// TwinCAT 3 PLC project Library
// Title: lcls-twincat-motion
// Company: SLAC
// ProjectVersion: 0.0.0
// ProgramVersion: 3.1.4026.17
// libraries:
//   LCLS General, * (SLAC)
//   lcls-twincat-math, * (SLAC - LCLS)
//   LCLS_OOPMotion, * (SLAC)
//   PMPS, * (SLAC - LCLS)
//   Tc2_EtherCAT, * (Beckhoff Automation GmbH)
//   Tc2_Math, * (Beckhoff Automation GmbH)
//   Tc2_MC2, * (Beckhoff Automation GmbH)
//   Tc2_Standard, * (Beckhoff Automation GmbH)
//   Tc2_System, * (Beckhoff Automation GmbH)
//   Tc2_Utilities, * (Beckhoff Automation GmbH)
//   Tc3_IPCDiag, * (Beckhoff Automation GmbH)
//   Tc3_JsonXml, * (Beckhoff Automation GmbH)
//   Tc3_Module, * (Beckhoff Automation GmbH)
//   TcUnit, * (www.tcunit.org)
// project tree:
//   DUTs/Deprecated/ ENUM_MotionRequest.TcDUT (not stored), DUT_MotionPneumaticActuator.TcDUT (not stored), DUT_MotionStage.TcDUT (not stored), DUT_PositionState.TcDUT (not stored), EL5042_Status.TcDUT (not stored), ENUM_EpicsHomeCmd.TcDUT (not stored), ENUM_EpicsInOut.TcDUT (not stored), ENUM_EpicsInOut_INT.TcDUT (not stored), ENUM_EpicsMotorCmd.TcDUT (not stored), ENUM_MotionFFType.TcDUT (not stored), ENUM_PnuematicActuatorPositionState.TcDUT (not stored), ENUM_StageBrakeMode.TcDUT (not stored), ENUM_StageEnableMode.TcDUT (not stored), ENUM_StatePMPSStatus.TcDUT (not stored)
//   DUTs/DS402/ ENUM_AxisStates.TcDUT (not stored), E_DS402DriveState.TcDUT (not stored), E_DS402EGU.TcDUT (not stored), E_DS402HomingMethod.TcDUT (not stored), E_DS402OpMode.TcDUT (not stored), E_HomeStates.TcDUT (not stored), E_Module.TcDUT (not stored), E_MoveMode.TcDUT (not stored), E_MoveState.TcDUT (not stored), ST_DS402Drive.TcDUT (not stored), ST_DS402DriveStatus.TcDUT (not stored)
//   DUTs/ E_EpicsHomeCmd.TcDUT (not stored), ST_AxisParameterSetExposed.TcDUT (not stored), E_LCLSMotionError.TcDUT (not stored), E_MotionFFType.TcDUT (not stored), E_StatePMPSStatus.TcDUT (not stored), ST_MotionEpicsInterface.TcDUT, ST_MotionStage.TcDUT (not stored), ST_PositionState.TcDUT (not stored), ST_StateEpicsToPlc.TcDUT (not stored), ST_StatePlcToEpics.TcDUT (not stored), ST_StatePMPSEpicsToPlc.TcDUT (not stored), ST_EL5042_Status.TcDUT (not stored), E_EpicsInOut.TcDUT (not stored), E_EpicsMotorCmd.TcDUT (not stored), E_MotionRequest.TcDUT (not stored), E_StageBrakeMode.TcDUT (not stored), E_StageEnableMode.TcDUT (not stored), ST_MotionPneumaticActuator.TcDUT (not stored), E_PnuematicActuatorPositionState.TcDUT (not stored), ST_RenishawAbsEnc.TcDUT (not stored), ST_StatePMPSPlcToEpics.TcDUT (not stored)
//   GVLs/ MOTION_GVL.TcGVL (not stored), MotionConstants.TcGVL (not stored)
//   / PlcTask.TcTTO (not stored)
//   POUs/Deprecated/ FB_EpicsInOut.TcPOU (not stored), FB_PositionStateBase.TcPOU (not stored), FB_PositionStateBase_WithPMPS.TcPOU (not stored), FB_PositionStateBase_WithPMPS_Test.TcPOU (not stored), FB_PositionStateInOut.TcPOU (not stored), FB_PositionStateInOut_WithPMPS.TcPOU (not stored), FB_PositionStateInOut_WithPMPS_Test.TcPOU (not stored), FB_PositionStateManager.TcPOU (not stored), FB_PositionStatePMPS.TcPOU (not stored), FB_PositionStatePMPS_Base.TcPOU (not stored), FB_PositionStatePMPS_Test.TcPOU (not stored), FB_StatePTPMove.TcPOU (not stored)
//   POUs/ImplicitChecks/ CheckBounds.TcPOU (not stored), CheckDivDInt.TcPOU (not stored), CheckDivLInt.TcPOU (not stored), CheckDivLReal.TcPOU (not stored), CheckDivReal.TcPOU (not stored)
//   POUs/Motion/DS402/ FB_MotionStageE727.TcPOU (not stored), FB_MotionStageMCS2.TcPOU (not stored), I_DS402GenericDrive.TcIO (not stored)
//   POUs/Motion/ FB_EncoderValue.TcPOU (not stored), FB_EncSaveRestore.TcPOU (not stored), FB_LogMotionError.TcPOU (not stored), FB_MotionBacklashCompensation.TcPOU (not stored), FB_MotionHoming.TcPOU (not stored), FB_MotionRequest.TcPOU (not stored), FB_MotionStage.TcPOU, FB_MotionStageNCParams.TcPOU (not stored), FB_MotionStageSim.TcPOU (not stored), FB_MotionPneumaticActuator.TcPOU (not stored), FB_MotionVirtualFrame.TcPOU (not stored)
//   POUs/Motion/Gantry/ FB_GantryAutoCoupling.TcPOU (not stored), FB_GantryDiffVirtualLimitSwitch.TcPOU (not stored)
//   POUs/Motion/PMPS/ FB_EncErrorFFO.TcPOU (not stored), FB_MiscStatesErrorFFO.TcPOU (not stored), FB_MotionBPTM.TcPOU (not stored), FB_MotionClearAsserts.TcPOU (not stored), FB_MotionReadPMPSDBND.TcPOU (not stored), FB_PerMotorFFOND.TcPOU (not stored), FB_NCErrorFFO.TcPOU (not stored), FB_PositionStatePMPS1D.TcPOU (not stored), FB_PositionStatePMPS2D.TcPOU (not stored), FB_PositionStatePMPS3D.TcPOU (not stored), FB_PositionStatePMPSND_Core.TcPOU (not stored), FB_Standard_PMPSDB.TcPOU (not stored), FB_StatePMPSEnables.TcPOU (not stored), FB_StatePMPSEnablesND.TcPOU (not stored)
//   POUs/Motion/States/Examples/ FB_PositionState1D_InOut.TcPOU (not stored), FB_PositionStatePMPS2D_InOut.TcPOU (not stored), FB_PositionStatePMPS1D_InOut.TcPOU (not stored), FB_PositionState2D_InOut.TcPOU (not stored)
//   POUs/Motion/States/ FB_PositionState2D.TcPOU (not stored), FB_PositionState3D.TcPOU (not stored), FB_PositionStateND_Core.TcPOU (not stored), FB_PositionStateMove.TcPOU (not stored), FB_PositionState1D.TcPOU (not stored), FB_PositionStateMoveND.TcPOU (not stored), FB_PositionStateRead.TcPOU (not stored), FB_PositionStateReadND.TcPOU (not stored), FB_StateSetupHelper.TcPOU (not stored), FB_StatesInputHandler.TcPOU (not stored)
//   POUs/Motion/States/Helpers/ FB_RawCountConverter.TcPOU (not stored), F_AtPositionState.TcPOU (not stored), F_PosOverLowerBound.TcPOU (not stored), F_PosUnderUpperBound.TcPOU (not stored), F_PosWithinDelta.TcPOU (not stored)
//   POUs/Motion/States/Internals/ FB_PositionStateInternal.TcPOU (not stored), FB_PositionStateInternalND.TcPOU (not stored), FB_PositionStateLock.TcPOU (not stored)
//   POUs/Motion/Utils/ FB_SetEnables.TcPOU (not stored), F_MotionErrorCodeLookup.TcPOU (not stored)
//   POUs/MotorTesting/ FB_MicroStepCountTest.TcPOU (not stored)
//   tc_mca_std_lib/DUTs/ DUT_AxisStatus_v0_01.TcDUT (not stored)
//   tc_mca_std_lib/GVLs/ GVL.TcGVL (not stored)
//   tc_mca_std_lib/POUs/ChangeConfig/ FB_ReadFloatParameter.TcPOU (not stored), FB_ReadParameterInNc_v1_00.TcPOU (not stored), FB_WriteFloatParameter.TcPOU (not stored), FB_WriteParameterInNc_v1_00.TcPOU (not stored)
//   tc_mca_std_lib/POUs/ErrorHandling/ DUT_ErrorState.TcDUT (not stored), DUT_TerminalError.TcDUT (not stored), FB_ErrorList.TcPOU (not stored), FB_TerminalError.TcPOU (not stored), GVL_ErrorSystem.TcGVL (not stored), ST_ErrorSystem.TcDUT (not stored)
//   tc_mca_std_lib/POUs/Hardware/EtherCAT_Terminals/Analog_Inputs/ EL3174_0002.TcPOU (not stored), EL3214.TcPOU (not stored), EL3255.TcPOU (not stored), FB_CalculateFrequency_3702_v0_01.TcPOU (not stored)
//   tc_mca_std_lib/POUs/Hardware/EtherCAT_Terminals/Digital_Inputs/ EL1008.TcPOU (not stored), EL1018.TcPOU (not stored), EL1808.TcPOU (not stored), EL1809.TcPOU (not stored), EL1819.TcPOU (not stored), FB_EL1252ASM_v1_00.TcPOU (not stored)
//   tc_mca_std_lib/POUs/Hardware/EtherCAT_Terminals/Digital_Outputs/ EL2014.TcPOU (not stored), EL2252.TcPOU (not stored), EL2808.TcPOU (not stored), EL2819.TcPOU (not stored)
//   tc_mca_std_lib/POUs/Hardware/EtherCAT_Terminals/Digital_Outputs/External_Types/ dutEL2521_Ctrl.TcDUT (not stored), dutEL2521_Status.TcDUT (not stored)
//   tc_mca_std_lib/POUs/Hardware/EtherCAT_Terminals/Measuring_Terminals/ EL5002.TcPOU (not stored), EL5021.TcPOU (not stored), EL5042.TcPOU (not stored), EL5101.TcPOU (not stored)
//   tc_mca_std_lib/POUs/Hardware/EtherCAT_Terminals/Motion/ EL7211_v1_00.TcPOU (not stored), EL9576_v1_00.TcPOU (not stored)
//   tc_mca_std_lib/POUs/Hardware/EtherCAT_Terminals/System/ EL9410.TcPOU (not stored), EL9505.TcPOU (not stored)
//   tc_mca_std_lib/POUs/Hardware/Other/ EK1200.TcPOU (not stored)
//   tc_mca_std_lib/POUs/Motion/ FB_DriveVirtual.TcPOU (not stored), FB_NcAxis.TcPOU (not stored)
//   tc_mca_std_lib/POUs/Motion/Homing/ FB_HomeDirect.TcPOU (not stored), FB_HomeFinish.TcPOU (not stored), FB_HomePrepare.TcPOU (not stored), FB_HomeReadNcVelocities.TcPOU (not stored), FB_HomeReadSoftLimEnable.TcPOU (not stored), FB_HomeToSwitch.TcPOU (not stored), FB_HomeVirtual.TcPOU (not stored), FB_HomeWriteNcVelocities.TcPOU (not stored), FB_HomeWriteSoftLimEnable.TcPOU (not stored)
//   Tests/ FB_AtPositionState_Test.TcPOU (not stored), FB_AxisParameterSetExposed_Test.TcPOU (not stored), FB_MiscStatesErrorFFO_Test.TcPOU (not stored), FB_MotionBPTM_Test.TcPOU (not stored), FB_MotionClearAsserts_Test.TcPOU (not stored), FB_MotionReadPMPSDBND_Test.TcPOU (not stored), FB_MotionVirtualFrame_Test.TcPOU (not stored), FB_NCErrorFFO_Test.TcPOU (not stored), FB_PerMotorFFOND_Test.TcPOU (not stored), FB_PositionStateMoveND_Test.TcPOU (not stored), FB_PositionStateMove_Test.TcPOU (not stored), FB_PositionStatePMPSND_Test.TcPOU (not stored), FB_PositionStateReadND_Test.TcPOU (not stored), FB_PositionStateRead_Test.TcPOU (not stored), FB_PositionStateND_Test.TcPOU (not stored), FB_PowerEnableMode_Test.TcPOU (not stored), FB_MotionBacklashCompensation_Test.TcPOU (not stored), FB_StatePMPSEnablesND_Test.TcPOU (not stored), FB_StatePMPSEnables_Test.TcPOU (not stored), FB_StateSetupHelper_Test.TcPOU (not stored), FB_TestHelperSetAndMove_Test.TcPOU (not stored), FB_TestStateInitTiming.TcPOU (not stored), PRG_TEST.TcPOU (not stored)
//   Tests/Helpers/ E_TestStates.TcDUT (not stored), FB_CauseNCError.TcPOU (not stored), FB_MotionStageSetAndMoveHelper.TcPOU (not stored), FB_MotionStageSetHelper.TcPOU (not stored), FB_MotorTestSuite.TcPOU (not stored), FB_PMPSJsonTestHelper.TcPOU (not stored), FB_TestHelperSetAndMove.TcPOU (not stored)

// ---- DUTs/ST_MotionEpicsInterface.TcDUT
TYPE ST_MotionEpicsInterface :
    // Defines the EPICS interface to moving a motor in TwinCAT
STRUCT
    // Name to use for log messages, fast faults, etc.
    sName: STRING;
    // Set to gantry difference tolerance
    nGantryTol: LINT:=0;
    // Encoder count at which this axis is aligned with other axis
    nEncRef: ULINT:=0;

    (* Commands *)
    // Used internally to request enables
    bEnable: BOOL;

    // Used internally to reset errors and other state
    {attribute 'pytmc' := '
        pv: PLC:bReset
        io: io
        field: ZNAM FALSE
        field: ONAM TRUE
        field: DESC Used internally to reset errors
    '}
    bReset: BOOL;
    // Used internally and by the IOC to start or stop a move
    bExecute: BOOL;

    (* Command Args *)
    // Used internally and by the IOC to pick what kind of move to do
    nCommand: INT;
    // Used internally and by the IOC to pass additional data to some commands
    nCmdData: INT;
    // Used internally and by the IOC to pick a destination for the move
    fPosition: LREAL;
    // Used internally and by the IOC to pick a move velocity
    fVelocity: LREAL;
    // Used internally and by the IOC to pick a move acceleration
    fAcceleration: LREAL;
    // Used internally and by the IOC to pick a move deceleration
    fDeceleration: LREAL;
    // Used internally and by the IOC to pick a home position
    {attribute 'pytmc' := '
        pv: PLC:fHomePosition
        io: io
        field: DESC Used internally and by the IOC to pick home position
    '}
    fHomePosition: LREAL;

    (* Info *)
    // Unique ID assigned to each axis in the NC
    nMotionAxisID: UDINT:=0;
    (* Returns *)
    // TRUE if in the middle of a command
    bBusy: BOOL;
    // TRUE if we've done a command and it has finished
    bDone: BOOL;
    // TRUE if the motor has been homed, or does not need to be homed
    bHomed: BOOL;

    // TRUE if we're in an error state
    {attribute 'pytmc' := '
        pv: PLC:bError
        io: i
        field: ZNAM FALSE
        field: ONAM TRUE
        field: DESC TRUE if we are in an error state
        update: 100Hz notify
    '}
    bError: BOOL;
    // Error code if nonzero
    {attribute 'pytmc' := '
        pv: PLC:nErrorId
        io: i
        field: DESC Error code if nonzero
        update: 100Hz notify
    '}
    nErrorId: UDINT;
    // Message to identify the error state
    {attribute 'pytmc' := '
        pv: PLC:sErrorMessage
        io: i
        field: DESC Message to identify the error state
        update: 100Hz notify
    '}
    sErrorMessage: STRING;

    // Misc axis status information for the IOC
    stAxisStatus: tc2_mc2.ST_AxisStatus;
END_STRUCT
END_TYPE

// ---- POUs/Motion/FB_MotionStage.TcPOU
FUNCTION_BLOCK FB_MotionStage IMPLEMENTS I_MotionStage
(*
    Default implementation for PLC behavior when motor IOC asks for a move
    This can be extended or replaced in your PLC project if you want
    non-default behavior to arise from the motor record processing
*)
VAR_IN_OUT
    stMotionStage: ST_MotionStage;
END_VAR
VAR
    fbDriveVirtual: FB_DriveVirtual;
    fbMotionHome: FB_MotionHoming;
    fbSaveRestore: FB_EncSaveRestore;
    fbLogError: FB_LogMotionError;
    fbBacklashCompensation: FB_MotionBacklashCompensation;
    bExecute: BOOL;
    bExecMove: BOOL;
    bExecHome: BOOL;
    bFwdHit: BOOL;
    bBwdHit: BOOL;
    ftExec: F_TRIG;
    rtExec: R_TRIG;
    rtUserExec: R_TRIG;
    rtTarget: R_TRIG;
    rtHomed: R_TRIG;
    fbSetEnables: FB_SetEnables;
    bPosGoal: BOOL;
    bNegGoal: BOOL;
    fbEncoderValue: FB_EncoderValue;
    fbNCParams: FB_MotionStageNCParams;
    bNewMoveReq: BOOL;
    bPrepareDisable: BOOL;
    bMoveCmd: BOOL;
    rtMoveCmdShortcut: R_TRIG;
    rtHomeCmdShortcut: R_TRIG;
    rtEnableMode: R_TRIG;

    {attribute 'pytmc' := 'pv: '}
    stMotionStatus : ST_MotionStatus;
    stMotionCmdPrev : ST_MotionCommand;
    {attribute 'pytmc' := 'pv: '}
    stMotionCmdNow : ST_MotionCommand;
    {attribute 'pytmc' := 'pv: '}
    stExMotionStatus : ST_ExtendedMotionStatus;
    stMotionStageMethods : REFERENCE TO ST_MotionStage;
END_VAR


stMotionStageMethods REF= stMotionStage;

IF NOT __ISVALIDREF(stMotionStage) THEN
    RETURN;
END_IF

// Main Motion Command Structure
IF stMotionCmdNow.bHalt <> stMotionCmdPrev.bHalt THEN
    stMotionStage.bExecute := NOT stMotionCmdNow.bHalt;
END_IF
IF stMotionCmdNow.bHomeCmd <> stMotionCmdPrev.bHomeCmd THEN
    stMotionStage.bHomeCmd := stMotionCmdNow.bHomeCmd;
END_IF
IF stMotionCmdNow.bMoveCmd <> stMotionCmdPrev.bMoveCmd THEN
    stMotionStage.bMoveCmd := stMotionCmdNow.bMoveCmd;
END_IF
IF stMotionCmdNow.bReset <> stMotionCmdPrev.bReset THEN
    stMotionStage.bReset := stMotionCmdNow.bReset;
END_IF
IF stMotionCmdNow.fAcceleration <> stMotionCmdPrev.fAcceleration THEN
    stMotionStage.fAcceleration := stMotionCmdNow.fAcceleration;
END_IF
IF stMotionCmdNow.fDeceleration <> stMotionCmdPrev.fDeceleration THEN
    stMotionStage.fDeceleration := stMotionCmdNow.fDeceleration;
END_IF
IF stMotionCmdNow.fHomePosition <> stMotionCmdPrev.fHomePosition THEN
    stMotionStage.fHomePosition := stMotionCmdNow.fHomePosition;
END_IF
IF stMotionCmdNow.fJerk <> stMotionCmdPrev.fJerk THEN
    //stMotionStage.fJerk := stMotionCmdNow.fJerk; NOT SUPPORTED BY THIS IMPLEMENTATION
END_IF
IF stMotionCmdNow.fPosition <> stMotionCmdPrev.fPosition THEN
    stMotionStage.fPosition := stMotionCmdNow.fPosition;
END_IF
IF stMotionCmdNow.fVelocity <> stMotionCmdPrev.fVelocity THEN
    stMotionStage.fVelocity := stMotionCmdNow.fVelocity;
END_IF
IF stMotionCmdNow.nCmdData <> stMotionCmdPrev.nCmdData THEN
    stMotionStage.nCmdData := stMotionCmdNow.nCmdData;
END_IF
IF stMotionCmdNow.nCommand <> stMotionCmdPrev.nCommand THEN
    stMotionStage.nCommand := stMotionCmdNow.nCommand;
END_IF

// Start with an accurate status
stMotionStage.Axis.ReadStatus();

// Check for the plc shortcut commands
// Used for testing or to circumvent motor record issues
rtMoveCmdShortcut(CLK:=stMotionStage.bMoveCmd);
rtHomeCmdShortcut(CLK:=stMotionStage.bHomeCmd);
// Execute on rising edge
IF rtMoveCmdShortcut.Q AND NOT stMotionStage.bExecute THEN
    stMotionStage.bExecute := TRUE;
    stMotionStage.nCommand := E_EpicsMotorCmd.MOVE_ABSOLUTE;

    // attempting to move an axis without homing first?
    IF stMotionStage.nHomingMode <> E_EpicsHomeCmd.NONE AND NOT stMotionStage.bHomed THEN
        // one can just set bHome here even though no homing was done?
        stMotionStage.sErrorMessage := 'Axis homing mode set, but homing routine pending';
    END_IF

ELSIF rtHomeCmdShortcut.Q AND NOT stMotionStage.bExecute THEN
    stMotionStage.bExecute := TRUE;
    stMotionStage.nCommand := E_EpicsMotorCmd.HOME;
END_IF
// Always reset, even if not rising edge, so command can be issued again
IF stMotionStage.bMoveCmd OR stMotionStage.bHomeCmd THEN
    stMotionStage.bMoveCmd := FALSE;
    stMotionStage.bHomeCmd := FALSE;
END_IF

// Automatically fill the correct nCmdData for homing
IF stMotionStage.nCommand = E_EpicsMotorCmd.HOME THEN
    stMotionStage.nCmdData := stMotionStage.nHomingMode;
END_IF

// Check if the command wants to cause a move
bMoveCmd R= stMotionStage.nCmdData = E_EpicsHomeCmd.ABSOLUTE_SET;
bMoveCmd R= stMotionStage.nCmdData = E_EpicsHomeCmd.NONE;
bMoveCmd S= stMotionStage.nCommand <> E_EpicsMotorCmd.HOME;

// Handle main execs
rtUserExec(CLK := stMotionStage.bExecute);
bNewMoveReq S= rtUserExec.Q AND bMoveCmd;
bNewMoveReq R= NOT stMotionStage.bExecute;
bPrepareDisable R= bNewMoveReq;

bPosGoal := stMotionStage.stAxisStatus.fActPosition < stMotionStage.fPosition;
bNegGoal := stMotionStage.stAxisStatus.fActPosition > stMotionStage.fPosition;

// Moves are automatically allowed if no safety hooks. Otherwise, some other code will set this.
stMotionStage.bSafetyReady S= stMotionStage.bPowerSelf;

// Transition to DURING_MOTION drive mode
rtEnableMode(CLK:=(stMotionStage.nEnableMode = E_StageEnableMode.DURING_MOTION));
// Handle auto-enable timing
CASE stMotionStage.nEnableMode OF
    E_StageEnableMode.ALWAYS:
        stMotionStage.bEnable := TRUE;
    E_StageEnableMode.DURING_MOTION:
        IF rtEnableMode.Q THEN
            stMotionStage.bEnable := FALSE;
        END_IF
        IF bNewMoveReq THEN
            IF stMotionStage.nCommand = E_EpicsMotorCmd.HOME THEN
                stMotionStage.bEnable := stMotionStage.bSafetyReady;
            ELSIF bPosGoal THEN
                IF stMotionStage.bAllForwardEnable THEN
                    stMotionStage.bEnable S= stMotionStage.bSafetyReady;
                ELSIF NOT stMotionStage.bError THEN
                    // Not an error, just a warning
                    stMotionStage.sErrorMessage := 'Cannot move past positive limit.';
                    stMotionStage.bExecute := FALSE;
                END_IF
            ELSIF bNegGoal THEN
                IF stMotionStage.bAllBackwardEnable THEN
                    stMotionStage.bEnable S= stMotionStage.bSafetyReady;
                ELSIF NOT stMotionStage.bError THEN
                    // Not an error, just a warning
                    stMotionStage.sErrorMessage := 'Cannot move past negative limit.';
                    stMotionStage.bExecute := FALSE;
                END_IF
            ELSE
                // Super rare condition where we asked for a move to exactly the same floating point we're already at
                stMotionStage.bEnable S= stMotionStage.bSafetyReady;
            END_IF
            IF stMotionStage.bEnable OR stMotionStage.bError THEN
                bNewMoveReq := FALSE;
            END_IF
        END_IF
END_CASE

// Update all enable booleans
fbSetEnables(stMotionStage:=stMotionStage);

IF stMotionStage.stAxisStatus.bBusy AND NOT bExecute THEN
    // Wait for the previous move to end
    bExecute := FALSE;
ELSIF bMoveCmd THEN
    // Do not start the move until we have power and the safety system says it is OK
    bExecute := stMotionStage.bExecute AND stMotionStage.bAllEnable AND stMotionStage.bEnableDone AND stMotionStage.bSafetyReady;
ELSE
    bExecute := stMotionStage.bExecute;
END_IF

IF bExecute AND NOT stMotionStage.bError THEN
    // Reset local warnings if things are going well
    stMotionStage.sErrorMessage := '';
END_IF

// No moves allowed in error states
IF stMotionStage.bError THEN
    bExecute := FALSE;
END_IF


bExecHome := bExecute AND stMotionStage.nCommand = 10;
bExecMove := bExecute AND NOT bExecHome;

// handles backlash compensention
fbBacklashCompensation(stMotionStage:=stMotionStage,
    bHoming:=bExecHome,
    bMoving:=bExecMove );

// Handle standard commands using ESS's FB
fbDriveVirtual(En:=TRUE,
    bEnable:=stMotionStage.bAllEnable,
    bReset:=stMotionStage.bReset,
    bExecute:=bExecMove,
    nCommand:=INT_TO_UINT(stMotionStage.nCommand),
    nCmdData:=INT_TO_UINT(stMotionStage.nCmdData),
    fVelocity:=stMotionStage.fVelocity,
    fPosition:=stMotionStage.fPosition,
    fAcceleration:=stMotionStage.fAcceleration,
    fDeceleration:=stMotionStage.fDeceleration,
    bLimitFwd:=stMotionStage.bAllForwardEnable,
    bLimitBwd:=stMotionStage.bAllBackwardEnable,
    bHomeSensor:=stMotionStage.bHome,
    fHomePosition:=stMotionStage.fHomePosition,
    bPowerSelf:=stMotionStage.bPowerSelf,
    nMotionAxisID=>stMotionStage.nMotionAxisID,
    Axis:=stMotionStage.Axis);

// Some custom home handling
fbMotionHome(
    stMotionStage:=stMotionStage,
    bExecute:=bExecHome);

// Update status again after the move starts or stops
stMotionStage.Axis.ReadStatus();

// Check for a new error
IF NOT stMotionStage.bError THEN
    stMotionStage.bError := fbDriveVirtual.bError;
    stMotionStage.nErrorId := fbDriveVirtual.nErrorId;
END_IF
IF NOT stMotionStage.bError THEN
    stMotionStage.bError := fbBacklashCompensation.bError;
    stMotionStage.nErrorId := fbBacklashCompensation.nErrorId;
END_IF
IF NOT stMotionStage.bError THEN
    stMotionStage.bError := fbMotionHome.bError;
    stMotionStage.nErrorId := fbMotionHome.nErrorId;
END_IF
IF NOT stMotionStage.bError AND stMotionStage.bExecute AND NOT stMotionStage.bUserEnable THEN
    stMotionStage.bError := TRUE;
    stMotionStage.nErrorId := 1;
    stMotionStage.sCustomErrorMessage := 'Move requested, but user enable is disabled!';
END_IF

// Set the error message if we have one
IF stMotionStage.bError THEN
    // Hook if other code wants to inject a non-NC error
    IF stMotionStage.sCustomErrorMessage <> '' THEN
        stMotionStage.sErrorMessage := stMotionSTage.sCustomErrorMessage;
    ELSE
        stMotionStage.sErrorMessage := F_MotionErrorCodeLookup(nErrorId := stMotionStage.nErrorId);
    END_IF
END_IF

fbLogError(
    stMotionStage:=stMotionStage,
    bEnable:=TRUE);

// When we start, set the busy/done appropriately
rtExec(CLK:=bExecute);
IF rtExec.Q THEN
    stMotionStage.bBusy := TRUE;
    stMotionStage.bDone := FALSE;
END_IF

// Force everything off in case of error
IF stMotionStage.bError THEN
    stMotionStage.bBusy := FALSE;
    stMotionStage.bDone := FALSE;
    stMotionStage.bEnable := FALSE;
END_IF

// Check the limits and cancel execution if appropriate. Without this block we have infinite error spam
bFwdHit := stMotionStage.Axis.Status.PositiveDirection AND NOT stMotionStage.bAllForwardEnable;
bBwdHit := stMotionStage.Axis.Status.NegativeDirection AND NOT stMotionStage.bAllBackwardEnable;
IF (bFwdHit OR bBwdHit) AND NOT fbMotionHome.bBusy THEN
    stMotionStage.bExecute := FALSE;
END_IF

// Check done moving via user stop, fbDriveVirtual and Target Position Monitoring, or from homing.
ftExec(CLK:=stMotionStage.bExecute);
rtTarget(CLK:=(stMotionStage.Axis.Status.InTargetPosition AND fbDriveVirtual.bDone AND bExecMove));
rtHomed(CLK:=fbMotionHome.bDone AND bExecHome);
IF ftExec.Q OR rtTarget.Q OR rtHomed.Q THEN
    IF NOT stMotionStage.bDone THEN
        stMotionStage.bDone := TRUE;
        stMotionStage.bBusy := FALSE;
        IF NOT stMotionStage.Axis.Status.Error THEN
            bExecute := FALSE;
            stMotionStage.bExecute := FALSE;
        END_IF
    END_IF
END_IF

// Handle auto-disable timing
bPrepareDisable S= stMotionStage.nEnableMode = E_StageEnableMode.DURING_MOTION AND ftExec.Q;
// Delay the disable until we reach standstill, else brake issues or other race conditions
IF bPrepareDisable AND stMotionStage.Axis.Status.MotionState = MC_AXISSTATE_STANDSTILL THEN
    bPrepareDisable := FALSE;
    stMotionStage.bEnable := FALSE;
END_IF

// Get a definitive bEnabled reading
CASE stMotionStage.Axis.Status.MotionState OF
    // We are not enabled if there is an issue
    MC_AXISSTATE_UNDEFINED, MC_AXISSTATE_DISABLED, MC_AXISSTATE_ERRORSTOP:
        stMotionStage.bEnableDone := FALSE;
    ELSE
        stMotionStage.bEnableDone := TRUE;
END_CASE

// Handle the brake. TRUE means brake disabled/released
IF stMotionStage.nBrakeMode <> E_StageBrakeMode.NO_BRAKE THEN
    CASE stMotionStage.Axis.Status.MotionState OF
        MC_AXISSTATE_UNDEFINED,
        MC_AXISSTATE_DISABLED,
        MC_AXISSTATE_ERRORSTOP:
            stMotionStage.bBrakeRelease := FALSE;
        MC_AXISSTATE_STANDSTILL:
            IF stMotionStage.nBrakeMode = E_StageBrakeMode.IF_MOVING THEN
                stMotionStage.bBrakeRelease := FALSE;
            ELSE
                stMotionStage.bBrakeRelease := TRUE;
            END_IF
        ELSE
            stMotionStage.bBrakeRelease := TRUE;
    END_CASE
END_IF

// Sync the epics status struct
stMotionStage.stAxisStatus := fbDriveVirtual.stAxisStatus;
stMotionStage.stAxisStatus.bEnabled := stMotionStage.bEnableDone;

// Override homing status, dmov as appropriate
stMotionStage.bHomed := fbMotionHome.bDone AND NOT fbMotionHome.bError;
stMotionStage.stAxisStatus.bHomed := stMotionStage.bHomed;
stMotionStage.stAxisStatus.bExecute := bExecute;
stMotionStage.stAxisStatus.nCommand := 3; // If this is not 3, the IOC stops updating positions during homing

// Fill in auxiliary status info
stMotionStage.fPosDiff := stMotionStage.Axis.NcToPlc.PosDiff;

// Reset everything when bReset is flagged
IF stMotionStage.bReset THEN
    stMotionStage.bEnable := FALSE;
    stMotionStage.bReset := FALSE;
    stMotionStage.bExecute := FALSE;
    stMotionStage.bError := FALSE;
    stMotionStage.nErrorId := 0;
    stMotionStage.sErrorMessage := '';
    stMotionStage.sCustomErrorMessage := '';
    bExecute := FALSE;
END_IF

fbEncoderValue(stMotionStage:=stMotionStage);
fbNCParams(
    stMotionStage:=stMotionStage,
    bEnable:=TRUE,
    tRefreshDelay:=T#1s);

// Save and restore as long as not an absolute encoder
fbSaveRestore(
    stMotionStage:=stMotionStage,
    bEnable:=stMotionStage.nHomingMode <> E_EpicsHomeCmd.NONE);

// Main Motion Status Structure
stMotionStatus.nMotionAxisID    := stMotionStage.Axis.NcToPlc.AxisId;
stMotionStatus.bEnabled         := stMotionStage.bAllEnable;
stMotionStatus.bHomeSensor      := stMotionStage.bHome;
stMotionStatus.bLimitBwd        := stMotionStage.bAllBackwardEnable;
stMotionStatus.bLimitFwd        := stMotionStage.bAllForwardEnable;
stMotionStatus.fActDiff         := stMotionStage.Axis.NcToPlc.PosDiff;
stMotionStatus.fActPosition     := stMotionStage.Axis.NcToPlc.ActPos;
stMotionStatus.fActVelocity     := stMotionStage.Axis.NcToPlc.ActVelo;
stMotionStatus.fOverride        := stMotionStage.Axis.PlcToNc.Override;
stMotionStatus.bBusy            := stMotionStage.bBusy;
stMotionStatus.bHomed           := stMotionStage.bHomed;
stMotionStatus.bWarning         := FALSE; // NOT SUPPORTED BY THIS IMPLEMENTATION
stMotionStatus.bError           := stMotionStage.bError;
stMotionStatus.nErrorId         := stMotionStage.nErrorId;
stMotionStatus.sErrorMessage    := stMotionStage.sErrorMessage;

// Extended Motion Status (Debug, Testing) NOT SUPPORTED BY THIS IMPLEMENTATION
// stExMotionStatus.bMotionAxisError
// stExMotionStatus.nMotionAxisErrorId
// stExMotionStatus.bInterlocksError
// stExMotionStatus.nInterlocksError
// stExMotionStatus.eDriveState
// stExMotionStatus.bAbortDone
// stExMotionStatus.bAborted
// stExMotionStatus.bLimHomeDone
// stExMotionStatus.bDriveWatchDogStatus
// stExMotionStatus.bNewMoveReq
// stExMotionStatus.bEnable
// stExMotionStatus.bIdling

// Main Motion Command Structure
stMotionCmdNow.bHalt := FALSE;
stMotionCmdNow.bHomeCmd := FALSE;
stMotionCmdNow.bMoveCmd := FALSE;
stMotionCmdNow.bReset := FALSE;
stMotionCmdNow.fAcceleration := stMotionStage.fAcceleration;
stMotionCmdNow.fDeceleration := stMotionStage.fDeceleration;
stMotionCmdNow.fHomePosition := stMotionStage.fHomePosition;
//stMotionCmdNow.fJerk := stMotionStage.fJerk; NOT SUPPORTED BY THIS IMPLEMENTATION
stMotionCmdNow.fPosition := stMotionStage.fPosition;
stMotionCmdNow.fVelocity := stMotionStage.fVelocity;
stMotionCmdNow.nCmdData := stMotionStage.nCmdData;
stMotionCmdNow.nCommand := stMotionStage.nCommand;

stMotionCmdPrev := stMotionCmdNow;


METHOD AbsoluteMove
VAR_INPUT
    Position	: LREAL;
    Velocity	: LREAL;
    Acceleration	: LREAL;
    Deceleration	: LREAL;
END_VAR

IF NOT __ISVALIDREF(THIS^.stMotionStageMethods) THEN
    RETURN;
END_IF

THIS^.stMotionStageMethods.fPosition := Position;
THIS^.stMotionStageMethods.fVelocity := Velocity;
THIS^.stMotionStageMethods.fAcceleration := Acceleration;
THIS^.stMotionStageMethods.fDeceleration := Deceleration;
THIS^.stMotionStageMethods.bMoveCmd := TRUE;
END_METHOD


METHOD AbsoluteMoveWithBacklashCompensation
VAR_INPUT
    Position	: LREAL;
    Velocity	: LREAL;
    Acceleration	: LREAL;
    Deceleration	: LREAL;
END_VAR

IF NOT __ISVALIDREF(THIS^.stMotionStageMethods) THEN
    RETURN;
END_IF

THIS^.stMotionStageMethods.fPosition := Position;
THIS^.stMotionStageMethods.fVelocity := Velocity;
THIS^.stMotionStageMethods.fAcceleration := Acceleration;
THIS^.stMotionStageMethods.fDeceleration := Deceleration;
THIS^.stMotionStageMethods.bMoveCmd := TRUE;
END_METHOD


PROPERTY BrakeMode : LCLS_OOPMotion.E_StageBrakeMode
GET

CASE THIS^.stMotionStageMethods.nBrakeMode OF
    E_StageBrakeMode.NO_BRAKE:
        BrakeMode := LCLS_OOPMotion.E_StageBrakeMode.NO_BRAKE;
    E_StageBrakeMode.IF_MOVING:
        BrakeMode := LCLS_OOPMotion.E_StageBrakeMode.IF_MOVING;
    E_StageBrakeMode.IF_ENABLED:
        BrakeMode := LCLS_OOPMotion.E_StageBrakeMode.IF_ENABLED;
END_CASE
END_GET
SET

CASE BrakeMode OF
    LCLS_OOPMotion.E_StageBrakeMode.NO_BRAKE:
        THIS^.stMotionStageMethods.nBrakeMode := E_StageBrakeMode.NO_BRAKE;
    LCLS_OOPMotion.E_StageBrakeMode.IF_MOVING:
        THIS^.stMotionStageMethods.nBrakeMode := E_StageBrakeMode.IF_MOVING;
    LCLS_OOPMotion.E_StageBrakeMode.IF_ENABLED:
        THIS^.stMotionStageMethods.nBrakeMode := E_StageBrakeMode.IF_ENABLED;
END_CASE
END_SET
END_PROPERTY


PROPERTY EnableMode : LCLS_OOPMotion.E_StageEnableMode
GET

CASE THIS^.stMotionStageMethods.nEnableMode OF
    E_StageEnableMode.ALWAYS:
        EnableMode := LCLS_OOPMotion.E_StageEnableMode.ALWAYS;
    E_StageEnableMode.DURING_MOTION:
        EnableMode := LCLS_OOPMotion.E_StageEnableMode.DURING_MOTION;
    E_StageEnableMode.NEVER:
        EnableMode := LCLS_OOPMotion.E_StageEnableMode.NEVER;
END_CASE
END_GET
SET

CASE EnableMode OF
    LCLS_OOPMotion.E_StageEnableMode.ALWAYS:
        THIS^.stMotionStageMethods.nEnableMode := E_StageEnableMode.ALWAYS;
    LCLS_OOPMotion.E_StageEnableMode.DURING_MOTION:
        THIS^.stMotionStageMethods.nEnableMode := E_StageEnableMode.DURING_MOTION;
    LCLS_OOPMotion.E_StageEnableMode.NEVER:
        THIS^.stMotionStageMethods.nEnableMode := E_StageEnableMode.NEVER;
END_CASE
END_SET
END_PROPERTY


PROPERTY ExMotionStatus : REFERENCE TO LCLS_OOPMotion.ST_ExtendedMotionStatus
GET

ExMotionStatus REF= THIS^.stExMotionStatus;
END_GET
END_PROPERTY


METHOD Halt

IF NOT __ISVALIDREF(THIS^.stMotionStageMethods) THEN
    RETURN;
END_IF

THIS^.stMotionStageMethods.bExecute := FALSE;
END_METHOD


METHOD Home
VAR_INPUT
    HomePosition	: LREAL;
    HomeMode	: INT;
END_VAR

IF NOT __ISVALIDREF(THIS^.stMotionStageMethods) THEN
    RETURN;
END_IF

THIS^.stMotionStageMethods.fHomePosition := HomePosition;

CASE HomeMode OF
    E_EpicsHomeCmd.ABSOLUTE_SET:
        THIS^.stMotionStageMethods.nHomingMode := E_EpicsHomeCmd.ABSOLUTE_SET;
    E_EpicsHomeCmd.AUTOZERO:
        THIS^.stMotionStageMethods.nHomingMode := E_EpicsHomeCmd.AUTOZERO;
    E_EpicsHomeCmd.CURRENT_POSITION_METHOD:
        THIS^.stMotionStageMethods.nHomingMode := E_EpicsHomeCmd.CURRENT_POSITION_METHOD;
    E_EpicsHomeCmd.HIGH_LIMIT:
        THIS^.stMotionStageMethods.nHomingMode := E_EpicsHomeCmd.HIGH_LIMIT;
    E_EpicsHomeCmd.HOME_VIA_HIGH:
        THIS^.stMotionStageMethods.nHomingMode := E_EpicsHomeCmd.HOME_VIA_HIGH;
    E_EpicsHomeCmd.HOME_VIA_LOW:
        THIS^.stMotionStageMethods.nHomingMode := E_EpicsHomeCmd.HOME_VIA_LOW;
    E_EpicsHomeCmd.LOW_LIMIT:
        THIS^.stMotionStageMethods.nHomingMode := E_EpicsHomeCmd.LOW_LIMIT;
    E_EpicsHomeCmd.NONE:
        THIS^.stMotionStageMethods.nHomingMode := E_EpicsHomeCmd.NONE;
END_CASE

THIS^.stMotionStageMethods.bHomeCmd := TRUE;
END_METHOD


PROPERTY MotionCmd : REFERENCE TO LCLS_OOPMotion.ST_MotionCommand
GET

MotionCmd REF= THIS^.stMotionCmdNow;
END_GET
END_PROPERTY


PROPERTY MotionStatus : REFERENCE TO LCLS_OOPMotion.ST_MotionStatus
GET

MotionStatus REF= THIS^.stMotionStatus;
END_GET
END_PROPERTY


METHOD Reset

IF NOT __ISVALIDREF(THIS^.stMotionStageMethods) THEN
    RETURN;
END_IF

THIS^.stMotionStageMethods.bReset := TRUE;
END_METHOD


PROPERTY SaveAxisParams : BOOL
SET

// NOT SUPPORTED BY THIS IMPLEMENTATION
END_SET
END_PROPERTY


METHOD StateMove
VAR_INPUT
    Execute	: BOOL;
END_VAR

IF NOT __ISVALIDREF(stMotionStageMethods) THEN
    RETURN;
END_IF
END_METHOD

END_FUNCTION_BLOCK
